// TIA Portal V20 export
FUNCTION "04 T4 LANT Transitions" : Void   // FC1412, LAD
TITLE = TRANSITIONS
{ S7_Optimized_Access := 'TRUE' }
// stored: AutoNumber false, SetENOAutomatically false
   VAR_TEMP
      Aux_real : Real;
   END_VAR
BEGIN

REGION Network 1: ============ TRANSITIONS ============
END_REGION

REGION Network 2: Transitions - Zone Status
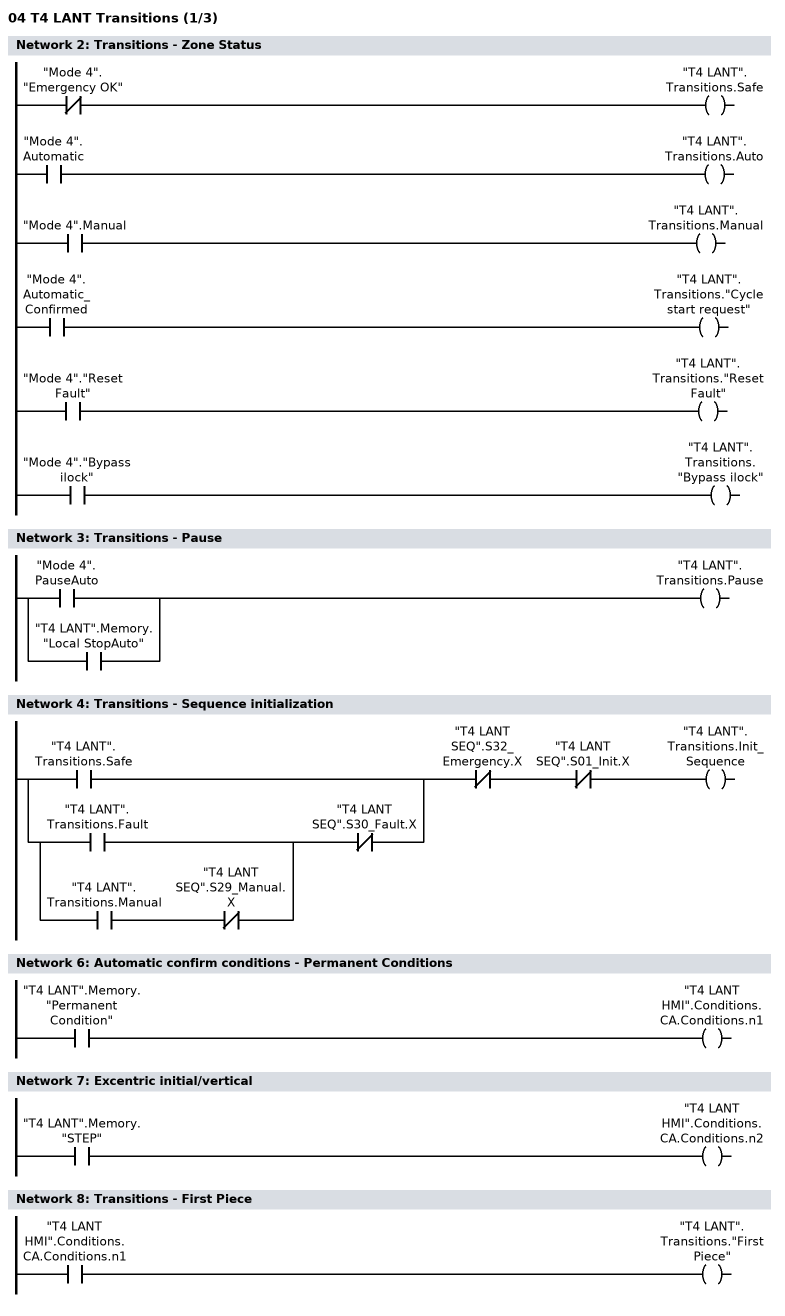
   RUNG wire#powerrail
      I_Contact( "Mode 4"."Emergency OK" )
      Coil( "T4 LANT".Transitions.Safe )
   END_RUNG
   RUNG wire#powerrail
      Contact( "Mode 4".Automatic )
      Coil( "T4 LANT".Transitions.Auto )
   END_RUNG
   RUNG wire#powerrail
      Contact( "Mode 4".Manual )
      Coil( "T4 LANT".Transitions.Manual )
   END_RUNG
   RUNG wire#powerrail
      Contact( "Mode 4".Automatic_Confirmed )
      Coil( "T4 LANT".Transitions."Cycle start request" )
   END_RUNG
   RUNG wire#powerrail
      Contact( "Mode 4"."Reset Fault" )
      Coil( "T4 LANT".Transitions."Reset Fault" )
   END_RUNG
   RUNG wire#powerrail
      Contact( "Mode 4"."Bypass ilock" )
      Coil( "T4 LANT".Transitions."Bypass ilock" )
   END_RUNG
   // the same network as SCL:
   "T4 LANT".Transitions.Safe := NOT "Mode 4"."Emergency OK";
   "T4 LANT".Transitions.Auto := "Mode 4".Automatic;
   "T4 LANT".Transitions.Manual := "Mode 4".Manual;
   "T4 LANT".Transitions."Cycle start request" := "Mode 4".Automatic_Confirmed;
   "T4 LANT".Transitions."Reset Fault" := "Mode 4"."Reset Fault";
   "T4 LANT".Transitions."Bypass ilock" := "Mode 4"."Bypass ilock";
END_REGION

REGION Network 3: Transitions - Pause
   RUNG wire#powerrail
      Contact( "Mode 4".PauseAuto )
      wire#w1
      Coil( "T4 LANT".Transitions.Pause )
   END_RUNG
   RUNG wire#powerrail
      Contact( "T4 LANT".Memory."Local StopAuto" )
   END_RUNG wire#w1
   // the same network as SCL:
   "T4 LANT".Transitions.Pause := "Mode 4".PauseAuto OR "T4 LANT".Memory."Local StopAuto";
END_REGION

REGION Network 4: Transitions - Sequence initialization
   RUNG wire#powerrail
      Contact( "T4 LANT".Transitions.Safe )
      wire#w1
      I_Contact( "T4 LANT SEQ".S32_Emergency.X )
      I_Contact( "T4 LANT SEQ".S01_Init.X )
      Coil( "T4 LANT".Transitions.Init_Sequence )
   END_RUNG
   RUNG wire#powerrail
      Contact( "T4 LANT".Transitions.Fault )
      wire#w2
      I_Contact( "T4 LANT SEQ".S30_Fault.X )
   END_RUNG wire#w1
   RUNG wire#powerrail
      Contact( "T4 LANT".Transitions.Manual )
      I_Contact( "T4 LANT SEQ".S29_Manual.X )
   END_RUNG wire#w2
   // the same network as SCL:
   "T4 LANT".Transitions.Init_Sequence := ("T4 LANT".Transitions.Safe OR (("T4 LANT".Transitions.Fault OR ("T4 LANT".Transitions.Manual AND NOT "T4 LANT SEQ".S29_Manual.X)) AND NOT "T4 LANT SEQ".S30_Fault.X)) AND NOT "T4 LANT SEQ".S32_Emergency.X AND NOT "T4 LANT SEQ".S01_Init.X;
END_REGION

REGION Network 5: ============ AUTOMATIC CONFIRM CONDITIONS - 1ST PIECE ============
END_REGION

REGION Network 6: Automatic confirm conditions - Permanent Conditions
   RUNG wire#powerrail
      Contact( "T4 LANT".Memory."Permanent Condition" )
      Coil( "T4 LANT HMI".Conditions.CA.Conditions.n1 )
   END_RUNG
   // the same network as SCL:
   "T4 LANT HMI".Conditions.CA.Conditions.n1 := "T4 LANT".Memory."Permanent Condition";
END_REGION

REGION Network 7: Excentric initial/vertical
   RUNG wire#powerrail
      Contact( "T4 LANT".Memory."STEP" )
      Coil( "T4 LANT HMI".Conditions.CA.Conditions.n2 )
   END_RUNG
   // the same network as SCL:
   "T4 LANT HMI".Conditions.CA.Conditions.n2 := "T4 LANT".Memory."STEP";
END_REGION

REGION Network 8: Transitions - First Piece
   RUNG wire#powerrail
      Contact( "T4 LANT HMI".Conditions.CA.Conditions.n1 )
      Coil( "T4 LANT".Transitions."First Piece" )
   END_RUNG
   // the same network as SCL:
   "T4 LANT".Transitions."First Piece" := "T4 LANT HMI".Conditions.CA.Conditions.n1;
END_REGION

REGION Network 9: Transitions - Piece presence
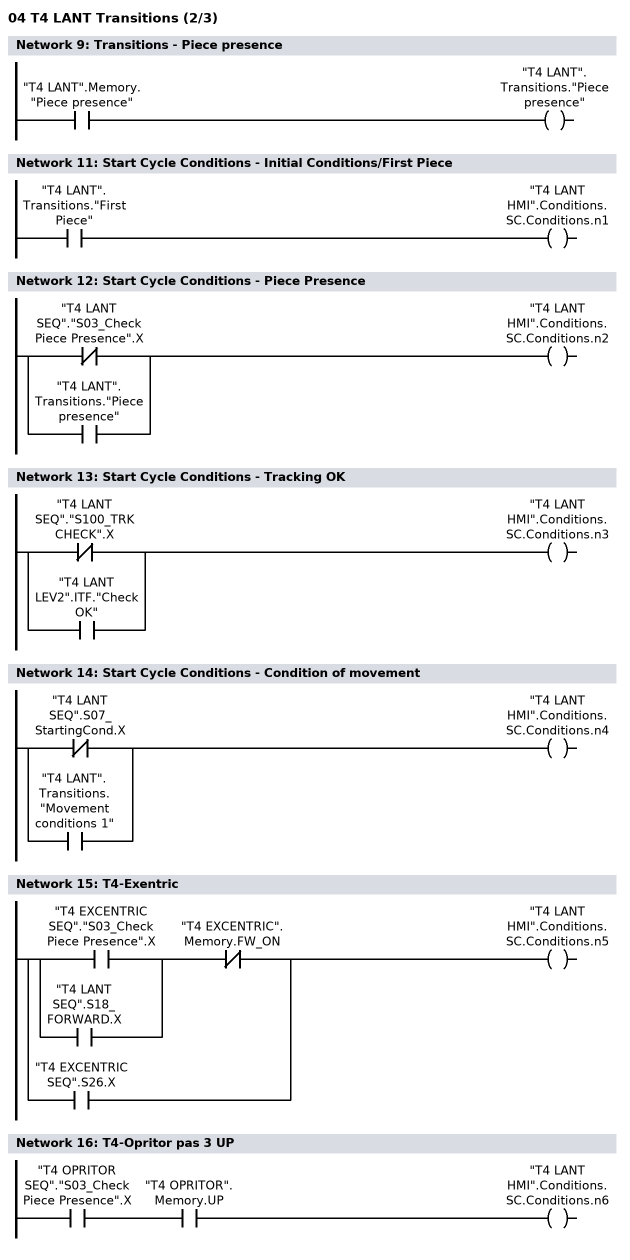
   RUNG wire#powerrail
      Contact( "T4 LANT".Memory."Piece presence" )
      Coil( "T4 LANT".Transitions."Piece presence" )
   END_RUNG
   // the same network as SCL:
   "T4 LANT".Transitions."Piece presence" := "T4 LANT".Memory."Piece presence";
END_REGION

REGION Network 10: ============ START CYCLE CONDITIONS ============
END_REGION

REGION Network 11: Start Cycle Conditions - Initial Conditions/First Piece
   RUNG wire#powerrail
      Contact( "T4 LANT".Transitions."First Piece" )
      Coil( "T4 LANT HMI".Conditions.SC.Conditions.n1 )
   END_RUNG
   // the same network as SCL:
   "T4 LANT HMI".Conditions.SC.Conditions.n1 := "T4 LANT".Transitions."First Piece";
END_REGION

REGION Network 12: Start Cycle Conditions - Piece Presence
   RUNG wire#powerrail
      I_Contact( "T4 LANT SEQ"."S03_Check Piece Presence".X )
      wire#w1
      Coil( "T4 LANT HMI".Conditions.SC.Conditions.n2 )
   END_RUNG
   RUNG wire#powerrail
      Contact( "T4 LANT".Transitions."Piece presence" )
   END_RUNG wire#w1
   // the same network as SCL:
   "T4 LANT HMI".Conditions.SC.Conditions.n2 := NOT "T4 LANT SEQ"."S03_Check Piece Presence".X OR "T4 LANT".Transitions."Piece presence";
END_REGION

REGION Network 13: Start Cycle Conditions - Tracking OK
   RUNG wire#powerrail
      I_Contact( "T4 LANT SEQ"."S100_TRK CHECK".X )
      wire#w1
      Coil( "T4 LANT HMI".Conditions.SC.Conditions.n3 )
   END_RUNG
   RUNG wire#powerrail
      Contact( "T4 LANT LEV2".ITF."Check OK" )
   END_RUNG wire#w1
   // the same network as SCL:
   "T4 LANT HMI".Conditions.SC.Conditions.n3 := NOT "T4 LANT SEQ"."S100_TRK CHECK".X OR "T4 LANT LEV2".ITF."Check OK";
END_REGION

REGION Network 14: Start Cycle Conditions - Condition of movement
   RUNG wire#powerrail
      I_Contact( "T4 LANT SEQ".S07_StartingCond.X )
      wire#w1
      Coil( "T4 LANT HMI".Conditions.SC.Conditions.n4 )
   END_RUNG
   RUNG wire#powerrail
      Contact( "T4 LANT".Transitions."Movement conditions 1" )
   END_RUNG wire#w1
   // the same network as SCL:
   "T4 LANT HMI".Conditions.SC.Conditions.n4 := NOT "T4 LANT SEQ".S07_StartingCond.X OR "T4 LANT".Transitions."Movement conditions 1";
END_REGION

REGION Network 15: T4-Exentric
   RUNG wire#powerrail
      Contact( "T4 EXCENTRIC SEQ"."S03_Check Piece Presence".X )
      wire#w1
      I_Contact( "T4 EXCENTRIC".Memory.FW_ON )
      wire#w2
      Coil( "T4 LANT HMI".Conditions.SC.Conditions.n5 )
   END_RUNG
   RUNG wire#powerrail
      Contact( "T4 LANT SEQ".S18_FORWARD.X )
   END_RUNG wire#w1
   RUNG wire#powerrail
      Contact( "T4 EXCENTRIC SEQ".S26.X )
   END_RUNG wire#w2
   // the same network as SCL:
   "T4 LANT HMI".Conditions.SC.Conditions.n5 := (("T4 EXCENTRIC SEQ"."S03_Check Piece Presence".X OR "T4 LANT SEQ".S18_FORWARD.X) AND NOT "T4 EXCENTRIC".Memory.FW_ON) OR "T4 EXCENTRIC SEQ".S26.X;
END_REGION

REGION Network 16: T4-Opritor pas 3 UP
   RUNG wire#powerrail
      Contact( "T4 OPRITOR SEQ"."S03_Check Piece Presence".X )
      Contact( "T4 OPRITOR".Memory.UP )
      Coil( "T4 LANT HMI".Conditions.SC.Conditions.n6 )
   END_RUNG
   // the same network as SCL:
   "T4 LANT HMI".Conditions.SC.Conditions.n6 := "T4 OPRITOR SEQ"."S03_Check Piece Presence".X AND "T4 OPRITOR".Memory.UP;
END_REGION

REGION Network 17: Transitions - Adjacent Machines
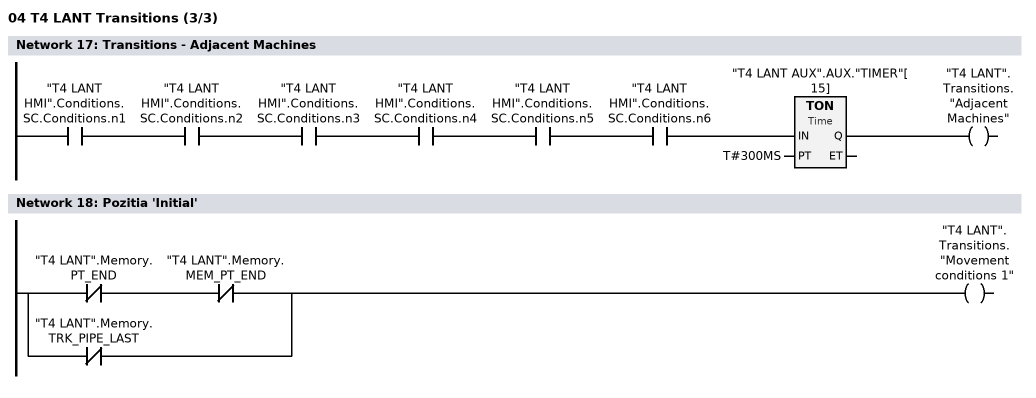
   RUNG wire#powerrail
      Contact( "T4 LANT HMI".Conditions.SC.Conditions.n1 )
      Contact( "T4 LANT HMI".Conditions.SC.Conditions.n2 )
      Contact( "T4 LANT HMI".Conditions.SC.Conditions.n3 )
      Contact( "T4 LANT HMI".Conditions.SC.Conditions.n4 )
      Contact( "T4 LANT HMI".Conditions.SC.Conditions.n5 )
      Contact( "T4 LANT HMI".Conditions.SC.Conditions.n6 )
      { S7_Templates := "time_type := Time" } "T4 LANT AUX".AUX."TIMER"[15].TON(pt := T#300MS, et =>)
      Coil( "T4 LANT".Transitions."Adjacent Machines" )
   END_RUNG
   // the same network as SCL:
   "T4 LANT AUX".AUX."TIMER"[15].TON(IN := "T4 LANT HMI".Conditions.SC.Conditions.n1 AND "T4 LANT HMI".Conditions.SC.Conditions.n2 AND "T4 LANT HMI".Conditions.SC.Conditions.n3 AND "T4 LANT HMI".Conditions.SC.Conditions.n4 AND "T4 LANT HMI".Conditions.SC.Conditions.n5 AND "T4 LANT HMI".Conditions.SC.Conditions.n6,
                           PT := T#300MS);
   "T4 LANT".Transitions."Adjacent Machines" := "T4 LANT AUX".AUX."TIMER"[15].Q;
END_REGION

REGION Network 18: Pozitia 'Initial'
   RUNG wire#powerrail
      I_Contact( "T4 LANT".Memory.PT_END )
      I_Contact( "T4 LANT".Memory.MEM_PT_END )
      wire#w1
      Coil( "T4 LANT".Transitions."Movement conditions 1" )
   END_RUNG
   RUNG wire#powerrail
      I_Contact( "T4 LANT".Memory.TRK_PIPE_LAST )
   END_RUNG wire#w1
   // the same network as SCL:
   "T4 LANT".Transitions."Movement conditions 1" := (NOT "T4 LANT".Memory.PT_END AND NOT "T4 LANT".Memory.MEM_PT_END) OR NOT "T4 LANT".Memory.TRK_PIPE_LAST;
END_REGION
END_FUNCTION
